PROGRAM MAIN
VAR
	FB_count:FB_count;
END_VAR

P_UPS();
systime();

IO_Link();
P_API_IO();
P_Modbus();
MAIN_ALarm();

P_Motion();
P_MediaTransport();
P_System();
P_InkSystem();
P_UVLed();
P_RollToRoll();
P_SpitUnit();
P_MaintenanceUnit();
P_SubTank();
P_TwinSAFE();


ACT_heart();



//IF VisuElems.CURRENTVISU='VIS_AXIS' THEN 
	//VisuElems.CURRENTVISU:='VIS_ISS';
//END_IF

ACTION ACT_heart:
FB_count(Add_Time:=T#0.1S , count=> GVL_API.count );
END_ACTION

END_PROGRAM

(* stored: Version 1.1.0.1, ProductVersion 3.1.4024.11
   POU MAIN: Id {d31199b4-3317-4917-a130-e2ee9bbfcd4b}, SpecialFunc None
   Action ACT_heart: Id {75ce6ba0-dae6-47b6-b9f5-85a3af4a56a2} *)
